TYPE stSettings_Rob EXTENDS stSettings_Base :
STRUCT
	
	LinearStandStillLimit : REAL := 1.0;	//mm/s
	AngularStandStillLimit : REAL := 0.001;	//rad/s
	
	UseSavedSecurePosition: BOOL := TRUE;
	NameOfSavedSecurePosition: STRING := 'SAFE';
	NameOfHomePosition: STRING := 'HOME';
	ManualSecurePosition: stJoint6;
	
	SafePositionTolerance: LREAL := 0.5;	//mm
	

	InstallationPose : ST_Pose; // BRF expressed in WRF : stVector3d
	StandardUnits : ST_StandardUnits := (
		Position            := eUnit.mm,
		Orientation         := eUnit.rad,
		Joint               := eUnit.rad,
		LinearVelocity      := eUnit.mm,
		AngularVelocity     := eUnit.rad,
		JointVelocity       := eUnit.rad,
		LinearAcceleration  := eUnit.mm,
		AngularAcceleration := eUnit.rad,
		JointAcceleration   := eUnit.rad
	); 	// Native unit standard of THIS robot. Subclasses overwrite in their declaration/FB_Init.
	// Base default = PLC standard (mm/rad), so conversions are a no-op if not overridden.
	HomingVelocity : REAL := 10; 		//mm/s
END_STRUCT
END_TYPE

(* stored: Version 1.1.0.1, ProductVersion 3.1.4026.18
   DUT stSettings_Rob: Id {255a0367-527b-4706-b91f-917c8b67132d} *)
